TYPE "UDT_STATUS_DETECTORES"
VERSION : 0.1
   STRUCT
      DTC01 : Bool;   // DETECTOR DE METAL 01 TC 06
      DTC02 : Bool;   // DETECTOR DE METAL 02 TC 12
      DTC03 : Bool;   // DETECTOR DE METAL 03 TC 16
   END_STRUCT;

END_TYPE

